/// Zeugwerk Application
PROGRAM ZModuleProgram
VAR_INPUT
{region "ZModuleProgram : Utility"}
  App : ZApp(displayName:='Zeugwerk-Application Template', com:=ZGlobal.Com.App);
  Datetime : ZAux.DateTimeUM;
  {attribute 'ZId' := ''}
{endregion}
{region "ZModuleProgram : Logging"}
  Alarming : ZApplication.Alarming(App, datetime := Datetime, com := ZGlobal.Com.Alarming);
  LoggerHmi : ZApplication.Messaging(App, datetime := Datetime, com := ZGlobal.Com.Messages);
  LoggerFile : ZAux.LoggerFile7FF(App, datetime := Datetime, filePath:='C:\Zeugwerk\logs\messages.log', target:='');
  Logger : ZAux.Logging;
  {attribute 'ZId' := ''}
{endregion}  
{attribute '__ZwPlcApplicationModuleProgramDeclaration__'} // Do not remove this attribute! It is used for code generation.
{region "PrimaryGear"}
{undefine RunInSeparateProgram}
{IF NOT (defined (PrimaryGear_disabled)) AND NOT (defined (RunInSeparateProgram))}
  PrimaryGear : GearUnit(name := 'PrimaryGear', // name of the unit (for logging)
					  parent := App, // caller of the Unit's cyclic method. If the Unit runs in its own context use 0
						configdata := ZGlobal.Data.Config.PrimaryGear,
						machinedata := ZGlobal.Data.Machine.PrimaryGear,
						calibrationdata := ZGlobal.Data.Calibration.PrimaryGear,
						com := ZGlobal.Com.Unit.PrimaryGear);
  {attribute 'section' := '__ZwPlcUnitProgramDeclaration__'}
  {attribute 'ZId' := 'd1deea68-6f8b-4ea5-9916-7be69dc951fa'}
{END_IF}
{endregion}
{region "Machine"}
{undefine RunInSeparateProgram}
{IF NOT (defined (Machine_disabled)) AND NOT (defined (RunInSeparateProgram))}
  Machine : MachineUnit(name := 'Machine', // name of the unit (for logging)
					  parent := App, // caller of the Unit's cyclic method. If the Unit runs in its own context use 0
						configdata := ZGlobal.Data.Config.Machine,
						machinedata := ZGlobal.Data.Machine.Machine,
						calibrationdata := ZGlobal.Data.Calibration.Machine,
						com := ZGlobal.Com.Unit.Machine);
  {attribute 'section' := '__ZwPlcUnitProgramDeclaration__'}
  {attribute 'ZId' := '9a1e8940-043c-4b8f-bd95-526fb267b71c'}
{END_IF}
{endregion}
{region "SimpleGear"}
{undefine RunInSeparateProgram}
{IF NOT (defined (SimpleGear_disabled)) AND NOT (defined (RunInSeparateProgram))}
  SimpleGear : GearUnit(name := 'SimpleGear', // name of the unit (for logging)
					  parent := App, // caller of the Unit's cyclic method. If the Unit runs in its own context use 0
						configdata := ZGlobal.Data.Config.SimpleGear,
						machinedata := ZGlobal.Data.Machine.SimpleGear,
						calibrationdata := ZGlobal.Data.Calibration.SimpleGear,
						com := ZGlobal.Com.Unit.SimpleGear);
  {attribute 'section' := '__ZwPlcUnitProgramDeclaration__'}
  {attribute 'ZId' := '215d1db4-d61a-4f46-91b5-612373b86c91'}
{END_IF}
{endregion}
{region "StruckigGear"}
{undefine RunInSeparateProgram}
{IF NOT (defined (StruckigGear_disabled)) AND NOT (defined (RunInSeparateProgram))}
  StruckigGear : GearUnit(name := 'StruckigGear', // name of the unit (for logging)
					  parent := App, // caller of the Unit's cyclic method. If the Unit runs in its own context use 0
						configdata := ZGlobal.Data.Config.StruckigGear,
						machinedata := ZGlobal.Data.Machine.StruckigGear,
						calibrationdata := ZGlobal.Data.Calibration.StruckigGear,
						com := ZGlobal.Com.Unit.StruckigGear);
  {attribute 'section' := '__ZwPlcUnitProgramDeclaration__'}
  {attribute 'ZId' := 'd827270e-999f-436d-80d5-b12442f5d1cf'}
{END_IF}
{endregion}
{attribute '__ZwPlcUnitProgramDeclaration__'} // Do not remove this attribute! It is used for code generation.
END_VAR

{region "ZModuleProgram : Utility"}
  Datetime.Cyclic();
  App.Cyclic();
  {attribute 'ZId' := ''}
{endregion}
{attribute '__ZwPlcApplicationModuleProgramImplementation__'} // Do not remove this attribute! It is used for code generation.

END_PROGRAM

(* stored: Version 1.1.0.1
   POU ZModuleProgram: Id {a120f957-5953-492b-ac4f-29b84ddfacdc}, SpecialFunc None *)
